// TIA Portal V17 export
// export: Created 2022-10-14T12:26:43.55541Z, ExportSetting WithDefaults, DisplayName Totally Integrated Automation Portal, DisplayVersion V17 Update 4, DisplayName TIA Portal Openness, DisplayVersion V17 Update 4, DisplayName TIA Portal Version Control Interface, DisplayVersion V17, DisplayName SINAMICS Startdrive Advanced, DisplayVersion V17 Update2, DisplayName SINAMICS Startdrive G130, G150, S120, S150, SINAMICS MV, S210, DisplayVersion V17 Update2, DisplayName SINAMICS Startdrive G110M, G120, G120C, G120D, G120P, G115D, DisplayVersion V17 Update2, DisplayName STEP 7 Professional, DisplayVersion V17 Update 4, DisplayName STEP 7 Safety, DisplayVersion V17, DisplayName WinCC Advanced / Unified PC, DisplayVersion V17 Update 4
DATA_BLOCK "1002_Device_iDB"   // DB1002
VERSION : 0.1
// stored: AutoNumber false, DBAccessibleFromOPCUA true, DBAccessibleFromWebserver true, InstanceOfName 1002_Device, InstanceOfType FB
"1002_Device"
   // VAR_INPUT
   //    Takt : Bool;
   //    HW_RCV : HW_SUBMODULE;
   //    HW_SND : HW_SUBMODULE;
   //    Addr : Array[1.."DeviceNr"] of Byte;
   //    Gruppen : Array[1.."DeviceNr"] of "Channels";
   //    "Message-Typ" : Byte;
   //    SubSysAdr : Byte;
   // END_VAR
   // VAR_OUTPUT
   //    Devices : Array[1.."DeviceNr"] of "Dates_Pro_Channel";
   // END_VAR
   // VAR
   //    HAdr { S7_SetPoint := 'True'} : Byte;
   //    HKanal : Byte;
   //    SND_ID : Byte;
   //    RCV_ID : Byte;
   //    Data_RCV : "RCV_Dates";
   //    i : Byte;
   //    K : Int;
   //    AA : Int;
   //    HM1 : Bool;
   //    HM2 : Bool;
   //    HM3 : Bool;
   //    HM4 : Bool;
   //    RESET_AA : Int;
   //    RESET_i : Int;
   //    RESET_i_Byte : USInt;
   // END_VAR
BEGIN
END_DATA_BLOCK
